// Mitsubishi GX Works2 project: ServMotor5   PLC: Q03UDV

PROGRAM MAIN
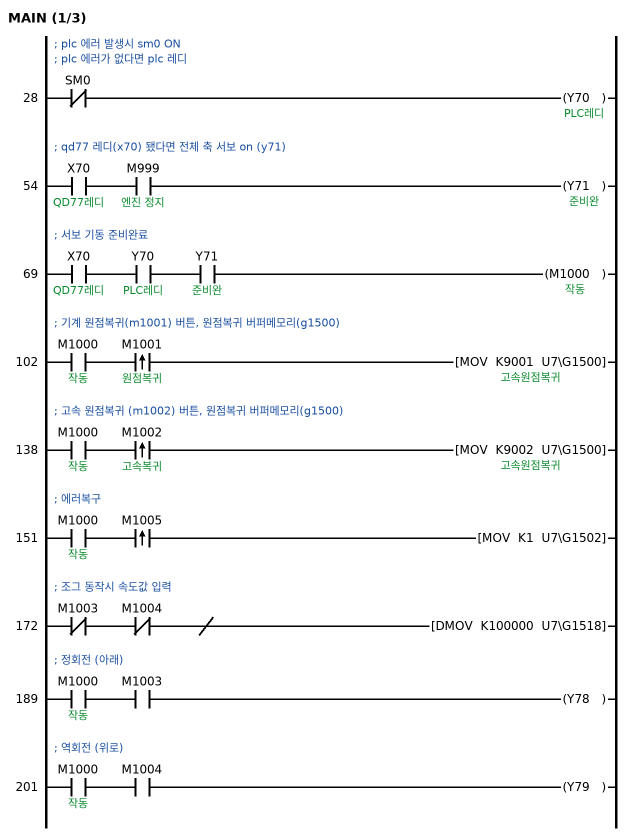
; plc 에러 발생시 sm0 ON
; plc 에러가 없다면 plc 레디
28    LDI     SM0
      OUT     Y70  ; PLC레디
; qd77 레디(x70) 됐다면 전체 축 서보 on (y71)
54    LD      X70  ; QD77레디
      AND     M999  ; 엔진 정지
      OUT     Y71  ; 준비완
; 서보 기동 준비완료
69    LD      X70  ; QD77레디
      AND     Y70  ; PLC레디
      AND     Y71  ; 준비완
      OUT     M1000  ; 작동
; 기계 원점복귀(m1001) 버튼, 원점복귀 버퍼메모리(g1500)
102   LD      M1000  ; 작동
      ANDP    M1001  ; 원점복귀
      MOV     K9001 U7\G1500  ; 고속원점복귀
; 고속 원점복귀 (m1002) 버튼, 원점복귀 버퍼메모리(g1500)
138   LD      M1000  ; 작동
      ANDP    M1002  ; 고속복귀
      MOV     K9002 U7\G1500
; 에러복구
151   LD      M1000  ; 작동
      ANDP    M1005
      MOV     K1 U7\G1502
; 조그 동작시 속도값 입력
172   LDI     M1003
      ANI     M1004
      INV
      DMOV    K100000 U7\G1518
; 정회전 (아래)
189   LD      M1000  ; 작동
      AND     M1003
      OUT     Y78
; 역회전 (위로)
201   LD      M1000  ; 작동
      AND     M1004
      OUT     Y79
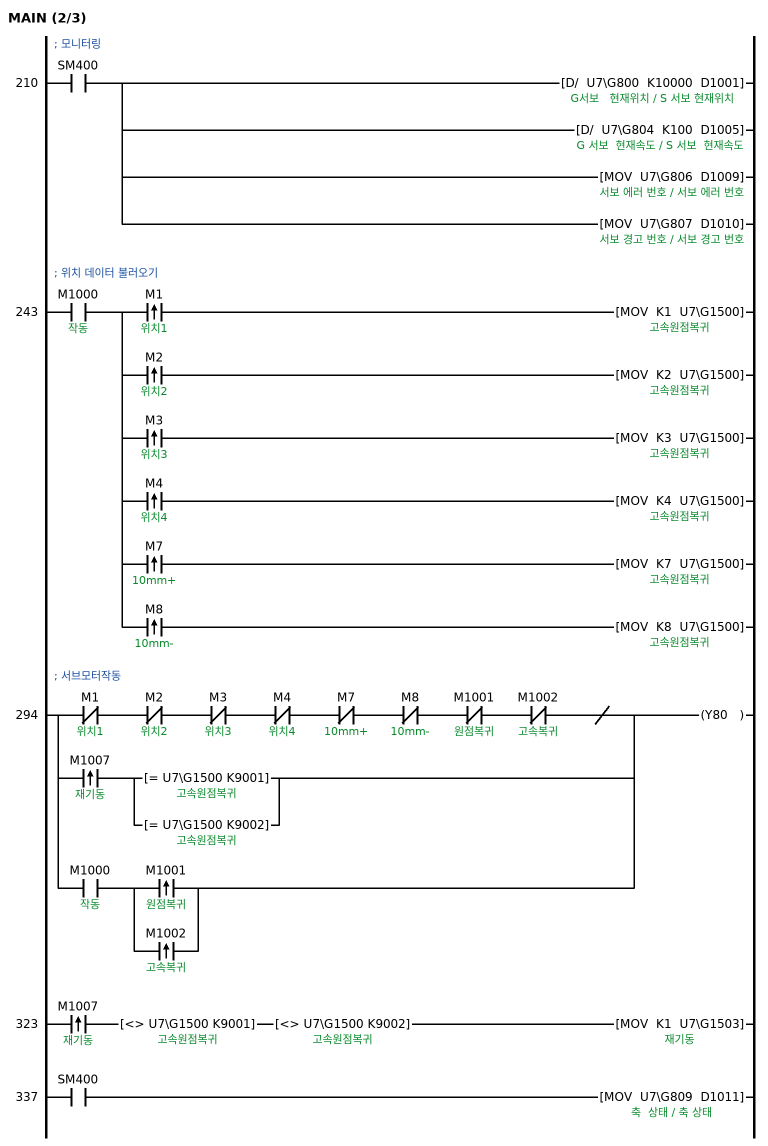
; 모니터링
210   LD      SM400
      D/      U7\G800 K10000 D1001  ; G서보   현재위치 / S 서보 현재위치
      D/      U7\G804 K100 D1005  ; G 서보  현재속도 / S 서보  현재속도
      MOV     U7\G806 D1009  ; 서보 에러 번호 / 서보 에러 번호
      MOV     U7\G807 D1010  ; 서보 경고 번호 / 서보 경고 번호
; 위치 데이터 불러오기
243   LD      M1000  ; 작동
      MPS
      ANDP    M1  ; 위치1
      MOV     K1 U7\G1500
      MRD
      ANDP    M2  ; 위치2
      MOV     K2 U7\G1500
      MRD
      ANDP    M3  ; 위치3
      MOV     K3 U7\G1500
      MRD
      ANDP    M4  ; 위치4
      MOV     K4 U7\G1500
      MRD
      ANDP    M7  ; 10mm+
      MOV     K7 U7\G1500
      MPP
      ANDP    M8  ; 10mm-
      MOV     K8 U7\G1500
; 서브모터작동
294   LDI     M1  ; 위치1
      ANI     M2  ; 위치2
      ANI     M3  ; 위치3
      ANI     M4  ; 위치4
      ANI     M7  ; 10mm+
      ANI     M8  ; 10mm-
      ANI     M1001  ; 원점복귀
      ANI     M1002  ; 고속복귀
      INV
      LDP     M1007  ; 재기동
      LD=     U7\G1500 K9001  ; 고속원점복귀
      OR=     U7\G1500 K9002  ; 고속원점복귀
      ANB
      ORB
      LD      M1000  ; 작동
      LDP     M1001  ; 원점복귀
      ORP     M1002  ; 고속복귀
      ANB
      ORB
      OUT     Y80
323   LDP     M1007  ; 재기동
      AND<>   U7\G1500 K9001  ; 고속원점복귀
      AND<>   U7\G1500 K9002  ; 고속원점복귀
      MOV     K1 U7\G1503  ; 재기동
337   LD      SM400
      MOV     U7\G809 D1011  ; 축  상태 / 축 상태
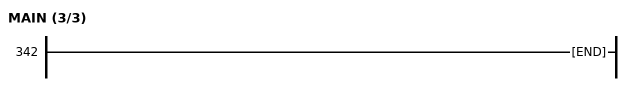
342   END
END_PROGRAM

// device comments not shown above
M1006  ; 축 정지
M1011  ; 축 상태
D1006  ; 서보 에러 번호
D1007  ; 서보 경고 번호
